(* PLC project  *)

CONFIGURATION PointTable_Data
END_CONFIGURATION
